// TIA Portal V19 export
DATA_BLOCK "Temperature Type_DB_2"   // DB12
// stored: InstanceOfName Temperature Type, InstanceOfType FB
"Temperature Type"
   // VAR_INPUT
   //    "RAW INPUT" : Int;
   //    "Scale MIN" : Real;
   //    "Scale MAX" : Real;
   // END_VAR
   // VAR_OUTPUT
   //    PV : Real;
   // END_VAR
   // VAR
   //    IEC_Timer_0_Instance_2 { S7_SetPoint := 'True'} : TON_TIME;
   //    IEC_Timer_0_Instance { S7_SetPoint := 'True'} : TOF_TIME;
   //    "INT TO REAL" : Real;
   // END_VAR
BEGIN
END_DATA_BLOCK
